{attribute 'GeneratedUsingTerminal: EL6201-0000-0017'}
{attribute addProperty BoxType "EL6201-0000-0017"}
{attribute addProperty Id "Slave_31A_DO0BOOL1Slave_31A_DO1BOOL1Slave_31A_DO2BOOL1Slave_31A_DO3BOOL1Slave_31B_DO0BOOL1Slave_31B_DO1BOOL1Slave_31B_DO2BOOL1Slave_31B_DO3BOOL1"}
{attribute addProperty CRC "3288739319"}
{attribute addProperty Size "8"}
TYPE Slave_31_Outputs_C4062DF7 :
STRUCT
	{attribute addProperty Name "Slave_31A_DO0"}
	Slave_31A_DO0 : BOOL;
	{attribute addProperty Name "Slave_31A_DO1"}
	Slave_31A_DO1 : BOOL;
	{attribute addProperty Name "Slave_31A_DO2"}
	Slave_31A_DO2 : BOOL;
	{attribute addProperty Name "Slave_31A_DO3"}
	Slave_31A_DO3 : BOOL;
	{attribute addProperty Name "Slave_31B_DO0"}
	Slave_31B_DO0 : BOOL;
	{attribute addProperty Name "Slave_31B_DO1"}
	Slave_31B_DO1 : BOOL;
	{attribute addProperty Name "Slave_31B_DO2"}
	Slave_31B_DO2 : BOOL;
	{attribute addProperty Name "Slave_31B_DO3"}
	Slave_31B_DO3 : BOOL;
END_STRUCT
END_TYPE

(* stored: Version 1.2.0.0, ProductVersion 3.1.4024.9
   DUT Slave_31_Outputs_C4062DF7: Id {5f51ae77-05ed-4a7f-8d56-d5ffdd70e96d} *)
